ABB RobotStudio station: ABB IRB140 robotkar - futószalag szimulátor.rspag

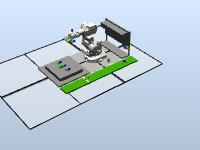
--- station ---
Station Solution3 (saved by RobotStudio format 3)
Controller IRB_140T_6kg_0.81m
  mechanical unit ROB_1: IRB140T_6_81_C_02, 6 joints, base frame (0, 0, 0) mm
Layout (positions relative to the parent item):
  - IRB140T_6_81_C_02 [mechanism, from Robots\IRB140T_6_81_C_G_02.rslib] at (0, 0, 0) mm; joint values [0, 0, 0, 0, 0.5236, 0] (rad or m)
  - Henger1 [part] at (700, 150, 96) mm, rotated rx 0 ry 0 rz 153.04 deg
  - Poz1 [part] at (-100, 50, 71) mm
  - Poz3 [part] at (-100, -50, 71) mm
  - SmatMefogo [smart component] at (506.29, 0, 679.5) mm, rotated rx 180 ry 60 rz 180 deg
      signals: DI Megfog, DI Elenged
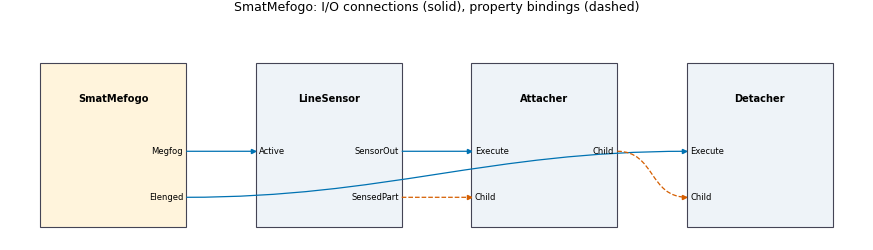
      connections:
        SmatMefogo.Megfog -> LineSensor.Active
        SmatMefogo.Elenged -> Detacher.Execute
        LineSensor.SensorOut -> Attacher.Execute
        LineSensor.SensedPart => Attacher.Child
        Attacher.Child => Detacher.Child
    - Megfogo [mechanism, from Libraries\Megfogo.rslib] at (0, 0, 0) mm, rotated rx 0 ry 0 rz -90 deg; joint values [0] (rad or m)
    - MegfogoTool [mechanism] at (0, 0, 0) mm
        TCP MyNewTool at (-15, 0, 70) mm, rotated rx -90 ry 0 rz -90 deg
        links: Dummy
    - LineSensor [smart component, from Components\LineSensor.rslib]
        properties: Start=[-0.0125 0.018 0.07]; End=[-0.0125 -0.019 0.07]; Radius=0.01; SensedPart=Hasab; SensedPoint=[0.764652587890625 0.0095 0.118910232543945]
      - _sensorPart_ [part]
    - Attacher [smart component, from Components\Attacher.rslib]
        properties: Parent=Megfogo; Flange=0; Child=Hasab; Mount=false; Offset=[0 0 0]; Orientation=[0 0 0]
    - Detacher [smart component, from Components\Detacher.rslib]
        properties: Child=Hasab; KeepPosition=true
  - SmartFSzalag [smart component] at (24.45, 0, 0) mm
      signals: DI Activate, DO SzalagErzekel
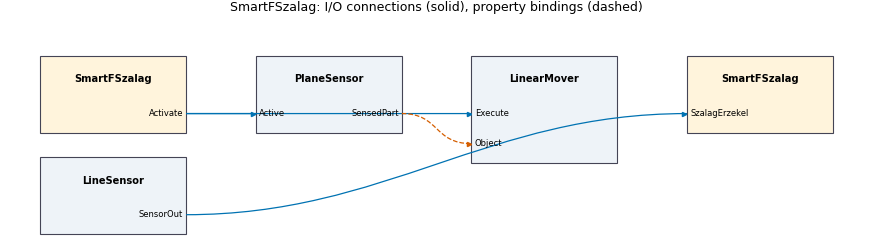
      connections:
        SmartFSzalag.Activate -> LinearMover.Execute
        SmartFSzalag.Activate -> PlaneSensor.Active
        LineSensor.SensorOut -> SmartFSzalag.SzalagErzekel
        PlaneSensor.SensedPart => LinearMover.Object
    - LinearMover [smart component, from Components\LinearMover.rslib]
        properties: Object=Hasab; Direction=[1 0 0]; Speed=0.1; Reference=Global; ReferenceObject=(none)
    - PlaneSensor [smart component, from Components\PlaneSensor.rslib]
        properties: Origin=[-0.7 0.425 0.027]; Axis1=[1.725 0 0]; Axis2=[0 0.2 0]; SensedPart=Hasab
      - _sensorPart_ [part]
    - FutoSzalag [part] at (-700, 425, 0) mm
    - LineSensor [smart component, from Components\LineSensor.rslib]
        properties: Start=[0.525 0.625 0.045]; End=[0.525 0.425 0.045]; Radius=0.005; SensedPart=(none); SensedPoint=[0 0 0]
      - _sensorPart_ [part]
  - Poz2 [part] at (-100, -100, 71) mm
  - Asztal [part]
  - Henger2 [part] at (700, -150, 96) mm
  - Henger3 [part] at (700, 0, 96) mm
  - Doboz [part, from Libraries\Doboz.rslib] at (434.43, -262.98, 25.91) mm
  - SolenoidValve [graphiccomponentgroup] at (400, -90, 651.5) mm, rotated rx 90 ry 0 rz 180 deg
    - coil_1 [part] at (16.04, 126.65, 10.8) mm, rotated rx 180 ry 0 rz -90 deg
    - coil_2 [part] at (16, -15.19, 10.52) mm, rotated rx 0 ry 0 rz 90 deg
    - solenoid [part]
  - Poz4 [part]
  - Hasab [part] at (0, 0, 0) mm
Attachment: SmatMefogo is attached to IRB140T_6_81_C_02 / Link6
Attachment: SolenoidValve is attached to IRB140T_6_81_C_02 / Link4
EventTableEntry 959: Group=, Trigger=DO10_1 960, Actions=[EventTableActionMechanicalPose 961], Comment=, ActivationMode=2, Cyclic=false
EventTableTriggerIO 960: IOValue=[1], IRC5Controller=? -1, Operator=0, SignalSource=IRB_140T_6kg_0.81m 463
EventTableActionMechanicalPose 961: VirtualSignal=, Mechanism=Megfogo 970, ToPoseName=Elenged, VirtualSignalValue=[1]
EventTableEntry 988: Group=, Trigger=DO10_2 989, Actions=[EventTableActionMechanicalPose 990], Comment=, ActivationMode=2, Cyclic=false
EventTableTriggerIO 989: IOValue=[1], IRC5Controller=? -1, Operator=0, SignalSource=IRB_140T_6kg_0.81m 463
EventTableActionMechanicalPose 990: VirtualSignal=, Mechanism=Megfogo 970, ToPoseName=Megfog, VirtualSignalValue=[1]
Collision set CollisionSet_1: FutoSzalag against Hasab, Henger1, Henger3, Henger2, near miss 0.01 m
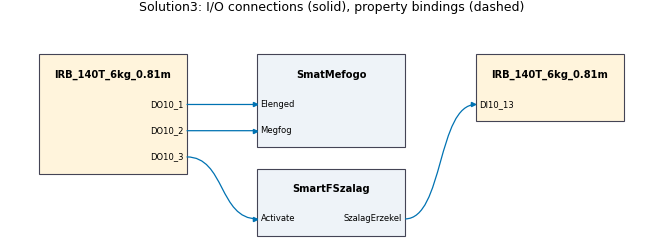
Station logic (signal -> signal, property => property):
  IRB_140T_6kg_0.81m.DO10_1 -> SmatMefogo.Elenged
  IRB_140T_6kg_0.81m.DO10_2 -> SmatMefogo.Megfog
  IRB_140T_6kg_0.81m.DO10_3 -> SmartFSzalag.Activate
  SmartFSzalag.SzalagErzekel -> IRB_140T_6kg_0.81m.DI10_13
Targets, tools, work objects and paths stored in the station and not in the controller backup, written as RAPID:
! task T_ROB1
MODULE Module1
  CONST robtarget FSz_vegefelett:=[[-438.059505293,555.460661011,365.486408927],[0.672643525,0.663438661,0.230130454,0.233323394],[1,-1,0,0],[9E9,9E9,9E9,9E9,9E9,9E9]];
ENDMODULE


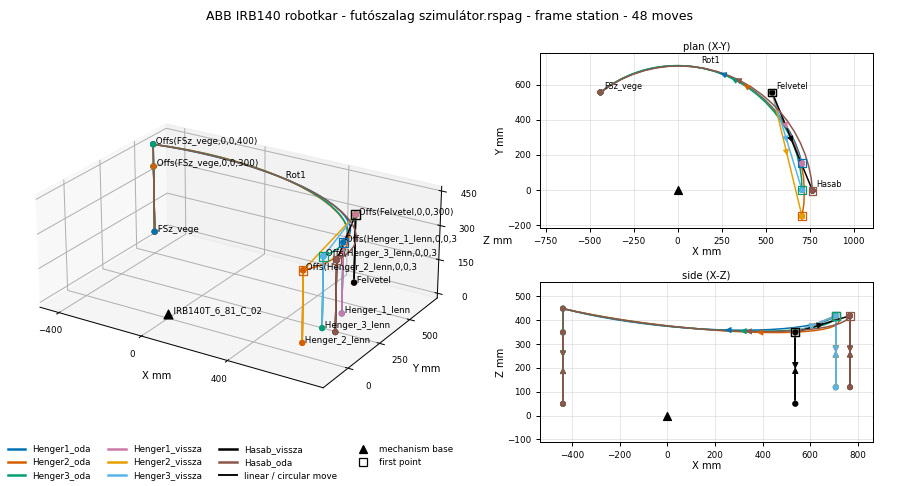
[picture p0: tool path of ABB IRB140 robotkar - futószalag szimulátor.rspag in frame station, 48 of 48 moves have a stored position in this frame; points joined in program order, loops and branches not executed]
--- Backups/IRB_140T_6kg_0.81m/RAPID/TASK1/PROGMOD/CalibData.mod ---
MODULE CalibData
	PERS tooldata MegfogoTool:=[TRUE,[[-15,0,70],[0.5,-0.5,0.5,-0.5]],[1,[0,0,1],[1,0,0,0],0,0,0]];
	PERS tooldata MyNewTool:=[TRUE,[[-15,0,70],[0.5,-0.5,0.5,-0.5]],[1,[0,0,1],[1,0,0,0],0,0,0]];
ENDMODULE

--- Backups/IRB_140T_6kg_0.81m/RAPID/TASK1/PROGMOD/Module1.mod ---
MODULE Module1
    CONST robtarget FSz_vege:=[[-438.059526577,555.460687999,48.955531046],[0.672643525,0.663438661,0.230130454,0.233323394],[1,-1,0,0],[9E9,9E9,9E9,9E9,9E9,9E9]];
    CONST robtarget Hasab:=[[767.152341031,-3.151777853,118.875787557],[0.503432685,0.496543913,-0.496543555,-0.503432391],[-1,-1,-1,0],[9E9,9E9,9E9,9E9,9E9,9E9]];
    CONST robtarget Henger_1_lenn:=[[707.41281816,151.613766479,118.875800346],[0.503432521,0.496543268,-0.496543664,-0.503433084],[0,0,0,0],[9E9,9E9,9E9,9E9,9E9,9E9]];
    CONST robtarget Henger_2_lenn:=[[707.4126997,-149.148355624,118.876093569],[0.503432871,0.496543143,-0.496543672,-0.503432849],[-1,-1,-1,0],[9E9,9E9,9E9,9E9,9E9,9E9]];
    CONST robtarget Henger_3_lenn:=[[707.412824643,0,118.87562894],[0.50343276,0.496543509,-0.496543509,-0.50343276],[-1,-1,-1,0],[9E9,9E9,9E9,9E9,9E9,9E9]];
    CONST robtarget Home:=[[463.138506398,0,576.806140488],[0.50343279,0.496543479,-0.496543479,-0.50343279],[-1,-1,-1,0],[9E9,9E9,9E9,9E9,9E9,9E9]];
    CONST robtarget Rot1:=[[110.910855884,698.664052428,365.486408927],[0.709756828,0.700044083,-0.055219241,-0.055985379],[0,-1,-1,0],[9E9,9E9,9E9,9E9,9E9,9E9]];
    CONST robtarget Felvetel:=[[537.334973477,554.640828476,49.574080385],[0.653372268,0.644431589,-0.278961189,-0.2828308],[0,0,0,0],[9E9,9E9,9E9,9E9,9E9,9E9]];
    PROC Megfog()
        PulseDO DO10_2;
        WaitTime 1;
    ENDPROC
    PROC Elenged()
        PulseDO DO10_1;
        WaitTime 1;
    ENDPROC
    PROC FutoszalagIndit()
        SetDO DO10_3, 1;
        WaitTime 1;
    ENDPROC
    PROC FutoszalagStop()
        SetDO DO10_3, 0;
        WaitTime 1;
    ENDPROC


PROC main()
       VAR num valasztas := -1;
       VAR num min := 0;
       VAR num max := 0;

       TPReadFK valasztas, "Hogy rakjon sorba?", "Novekvo", "Csokkeno","","","";
       IF(valasztas = 1) THEN
           IF(max=0 AND min=0) THEN
                max:=1;


                Henger1_oda;
                Futoszalag;
                Henger2_oda;
                Henger1_vissza;
                Futoszalag;
                Henger3_oda;
                Henger3_vissza;
                Futoszalag;
                Hasab_oda;
                Henger2_vissza;
                Futoszalag;
                Hasab_vissza;


           ELSEIF max = 1 THEN
                max:=1;
                min:=0;


                Henger1_oda;
                Futoszalag;
                Henger3_oda;
                Henger1_vissza;
                Futoszalag;
                Henger2_oda;
                Henger3_vissza;
                Futoszalag;
                Hasab_oda;
                Henger2_vissza;
                Futoszalag;
                Hasab_vissza;


           ELSEIF min = 1 THEN
                max:=1;
                min:=0;


                Henger1_oda;
                Futoszalag;
                Hasab_oda;
                Hasab_vissza;
                Futoszalag;
                Henger2_oda;
                Henger2_vissza;
                Futoszalag;
                Henger3_oda;
                Henger3_vissza;
                Futoszalag;
                Henger1_vissza;


           ENDIF
       ELSEIF valasztas = 2 THEN
           IF(max=0 AND min=0) THEN
                min:=1;


                Hasab_oda;
                Futoszalag;
                Henger1_oda;
                Henger1_vissza;
                Futoszalag;
                Henger3_oda;
                Hasab_vissza;
                Futoszalag;
                Henger2_oda;
                Henger3_vissza;
                Futoszalag;
                Henger2_vissza;


           ELSEIF max = 1 THEN
                max:=0;
                min:=1;


                Hasab_oda;
                Futoszalag;
                Henger1_oda;
                Henger1_vissza;
                Futoszalag;
                Henger2_oda;
                Hasab_vissza;
                Futoszalag;
                Henger3_oda;
                Henger3_vissza;
                Futoszalag;
                Henger2_vissza;


           ELSEIF min = 1 THEN
                max:=0;
                min:=1;


                Henger1_oda;
                Futoszalag;
                Henger3_oda;
                Henger1_vissza;
                Futoszalag;
                Henger2_oda;
                Henger3_vissza;
                Futoszalag;
                Hasab_oda;
                Henger2_vissza;
                Futoszalag;
                Hasab_vissza;



           ENDIF
       ENDIF
    ENDPROC


    PROC Henger1_oda()
        MoveL Offs(Henger_1_lenn,0,0,300),v200,fine,MegfogoTool\WObj:=wobj0;
        MoveL Henger_1_lenn,v200,fine,MegfogoTool\WObj:=wobj0;
        Megfog;
        WaitTime 1;
        MoveL Offs(Henger_1_lenn,0,0,300),v200,fine,MegfogoTool\WObj:=wobj0;
        MoveC Rot1,Offs(FSz_vege,0,0,400),v200,fine,MegfogoTool\WObj:=wobj0;
        MoveL FSz_vege, v200,fine,MegfogoTool\WObj:=wobj0;
        Elenged;
        WaitTime 1;
        MoveL Offs(FSz_vege,0,0,300),v200,fine,MegfogoTool\WObj:=wobj0;
    ENDPROC

    PROC Henger2_oda()
        MoveL Offs(Henger_2_lenn,0,0,300),v200,fine,MegfogoTool\WObj:=wobj0;
        MoveL Henger_2_lenn,v200,fine,MegfogoTool\WObj:=wobj0;
        Megfog;
        WaitTime 1;
        MoveL Offs(Henger_2_lenn,0,0,300),v200,fine,MegfogoTool\WObj:=wobj0;
        MoveC Rot1,Offs(FSz_vege,0,0,400),v200,fine,MegfogoTool\WObj:=wobj0;
        MoveL FSz_vege,v200,fine,MegfogoTool\WObj:=wobj0;
        Elenged;
        WaitTime 1;
        MoveL Offs(FSz_vege,0,0,300),v200,fine,MegfogoTool\WObj:=wobj0;
    ENDPROC

    PROC Henger3_oda()
        MoveL Offs(Henger_3_lenn,0,0,300),v200,fine,MegfogoTool\WObj:=wobj0;
        MoveL Henger_3_lenn,v200,fine,MegfogoTool\WObj:=wobj0;
        Megfog;
        WaitTime 1;
        MoveL Offs(Henger_3_lenn,0,0,300),v200,fine,MegfogoTool\WObj:=wobj0;
        MoveC Rot1,Offs(FSz_vege,0,0,400),v200,fine,MegfogoTool\WObj:=wobj0;
        MoveL FSz_vege,v200,fine,MegfogoTool\WObj:=wobj0;
        Elenged;
        WaitTime 1;
        MoveL Offs(FSz_vege,0,0,300),v200,fine,MegfogoTool\WObj:=wobj0;
    ENDPROC

    PROC Henger1_vissza()
        MoveL Offs(Felvetel,0,0,300),v200,fine,MegfogoTool\WObj:=wobj0;
        MoveL Felvetel,v200,fine,MegfogoTool\WObj:=wobj0;
        Megfog;
        WaitTime 1;
        MoveL Offs(Felvetel,0,0,300),v200,fine,MegfogoTool\WObj:=wobj0;
        MoveL Offs(Henger_1_lenn,0,0,300),v200,fine,MegfogoTool\WObj:=wobj0;
        MoveL Henger_1_lenn,v200,fine,MegfogoTool\WObj:=wobj0;
        Elenged;
        WaitTime 1;
        MoveL Offs(Henger_1_lenn,0,0,300),v200,fine,MegfogoTool\WObj:=wobj0;
    ENDPROC

    PROC Henger2_vissza()
        MoveL Offs(Felvetel,0,0,300),v200,fine,MegfogoTool\WObj:=wobj0;
        MoveL Felvetel,v200,fine,MegfogoTool\WObj:=wobj0;
        Megfog;
        WaitTime 1;
        MoveL Offs(Felvetel,0,0,300),v200,fine,MegfogoTool\WObj:=wobj0;
        MoveL Offs(Henger_2_lenn,0,0,300),v200,fine,MegfogoTool\WObj:=wobj0;
        MoveL Henger_2_lenn,v200,fine,MegfogoTool\WObj:=wobj0;
        Elenged;
        WaitTime 1;
        MoveL Offs(Henger_2_lenn,0,0,300),v200,fine,MegfogoTool\WObj:=wobj0;
    ENDPROC

    PROC Henger3_vissza()
        MoveL Offs(Felvetel,0,0,300),v200,fine,MegfogoTool\WObj:=wobj0;
        MoveL Felvetel,v200,fine,MegfogoTool\WObj:=wobj0;
        Megfog;
        WaitTime 1;
        MoveL Offs(Felvetel,0,0,300),v200,fine,MegfogoTool\WObj:=wobj0;
        MoveL Offs(Henger_3_lenn,0,0,300),v200,fine,MegfogoTool\WObj:=wobj0;
        MoveL Henger_3_lenn,v200,fine,MegfogoTool\WObj:=wobj0;
        Elenged;
        WaitTime 1;
        MoveL Offs(Henger_3_lenn,0,0,300),v200,fine,MegfogoTool\WObj:=wobj0;
    ENDPROC

    PROC Hasab_vissza()
        MoveL Offs(Felvetel,0,0,300),v200,fine,MegfogoTool\WObj:=wobj0;
        MoveL Felvetel,v200,fine,MegfogoTool\WObj:=wobj0;
        Megfog;
        WaitTime 1;
        MoveL Offs(Felvetel,0,0,300),v200,fine,MegfogoTool\WObj:=wobj0;
        MoveL Offs(Hasab,0,0,300),v200,fine,MegfogoTool\WObj:=wobj0;
        MoveL Hasab,v200,fine,MegfogoTool\WObj:=wobj0;
        Elenged;
        WaitTime 1;
        MoveL Offs(Hasab,0,0,300),v200,fine,MegfogoTool\WObj:=wobj0;
    ENDPROC

    PROC Hasab_oda()
        MoveL Offs(Hasab,0,0,300),v200,fine,MegfogoTool\WObj:=wobj0;
        MoveL Hasab,v200,fine,MegfogoTool\WObj:=wobj0;
        Megfog;
        WaitTime 1;
        MoveL Offs(Hasab,0,0,300),v200,fine,MegfogoTool\WObj:=wobj0;
        MoveC Rot1,Offs(FSz_vege,0,0,400),v200,fine,MegfogoTool\WObj:=wobj0;
        MoveL FSz_vege,v200,fine,MegfogoTool\WObj:=wobj0;
        Elenged;
        WaitTime 1;
        MoveL Offs(FSz_vege,0,0,300),v200,fine,MegfogoTool\WObj:=wobj0;
    ENDPROC

  PROC Futoszalag()
        FutoszalagIndit;
        WaitDI DI10_13,1;
        FutoszalagStop;
    ENDPROC


ENDMODULE

--- Backups/IRB_140T_6kg_0.81m/RAPID/TASK1/SYSMOD/LINKEDM.sys ---
%%%
  VERSION:1
  LANGUAGE:ENGLISH
%%%

MODULE LINKEDM (SYSMODULE)

! FOLLOWER
!     Name of electronically linked follower axis used by operator at teach pendent.
      PERS string l_f_axis_name{5}       :=  ["",  "", "", "", ""];

!     Name of the mechanical unit for follower axis.
      PERS string l_f_mecunt_n{5}  :=  ["", "", "", "", ""];

!     Linked follower axis number in the mechanical unit (first axis in mech. unit is number 1).
      PERS num l_f_axis_no{5}      :=  [0,          0,   0,  0,  0];

! MASTER
!     Name of the mechanical unit for linked master axis.
      PERS string l_m_mecunt_n{5} :=  ["", "", "", "", ""];

!     Linked master axis number in the mechanical unit (first axis in mech. unit is number 1).
!     See axis number table in documentation for different master mechanical units.
      PERS num l_m_axis_no{5}     :=  [0,  0,  0,  0,  0];

! POSITION OFFSET
!     The increase of the allowed offset position between the master and follower
!     positions, used when starting AUTO mode. As soon as the offset is decreased
!     the old configurated parameter is used.
!     Example: 3 => the configurated value of allowed offset is increased 3 times.
      PERS num offset_ratio{5}       :=  [10,  10,   10,  10,  10];

! SPEED RATIO
!     Speed_ratio used in AUTO and JOG modes [ very_slow   slow    normal    fast]
!     Value 1 = max allowed manual speed.
      CONST num speed_ratio {20}      := [0.01, 0.01, 0.01, 0.01, 0.01,
                                          0.05, 0.05, 0.05, 0.05, 0.05,
                                          0.20, 0.20, 0.20, 0.20, 0.20,
                                          1.00, 1.00, 1.00, 1.00, 1.00];

! STEP SIZE
!     Displacement position used in JOG mode for each activation of positive or
!     negative movement.                  [very_short    short   normal   long]
!     Unit degees or meter.
      CONST num displacement {20}     := [0.001, 0.001, 0.001, 0.001, 0.001,
                                          0.005, 0.005, 0.005, 0.005, 0.005,
                                          0.020, 0.020, 0.020, 0.020, 0.020,
                                          0.100, 0.100, 0.100, 0.100, 0.100];


!-------------------------------------------------------------
 PROC Linked_m ()
      Linked_m_exe ;
 ENDPROC
ENDMODULE

--- Backups/IRB_140T_6kg_0.81m/SYSPAR/EIO.cfg ---
EIO:CFG_1.0:6:0::
#
EIO_SIGNAL:

      -Name "DO10_1" -SignalType "DO" -Access "All"

      -Name "DO10_2" -SignalType "DO" -Access "All"

      -Name "DO10_3" -SignalType "DO" -Access "All"

      -Name "DI10_13" -SignalType "DI" -Access "All"
